// SIMATIC S7-200 project (STEP 7-Micro/WIN), CPU 224XP REL 02.01

ORGANIZATION_BLOCK 主程序:OB1
TITLE=程序注释
BEGIN
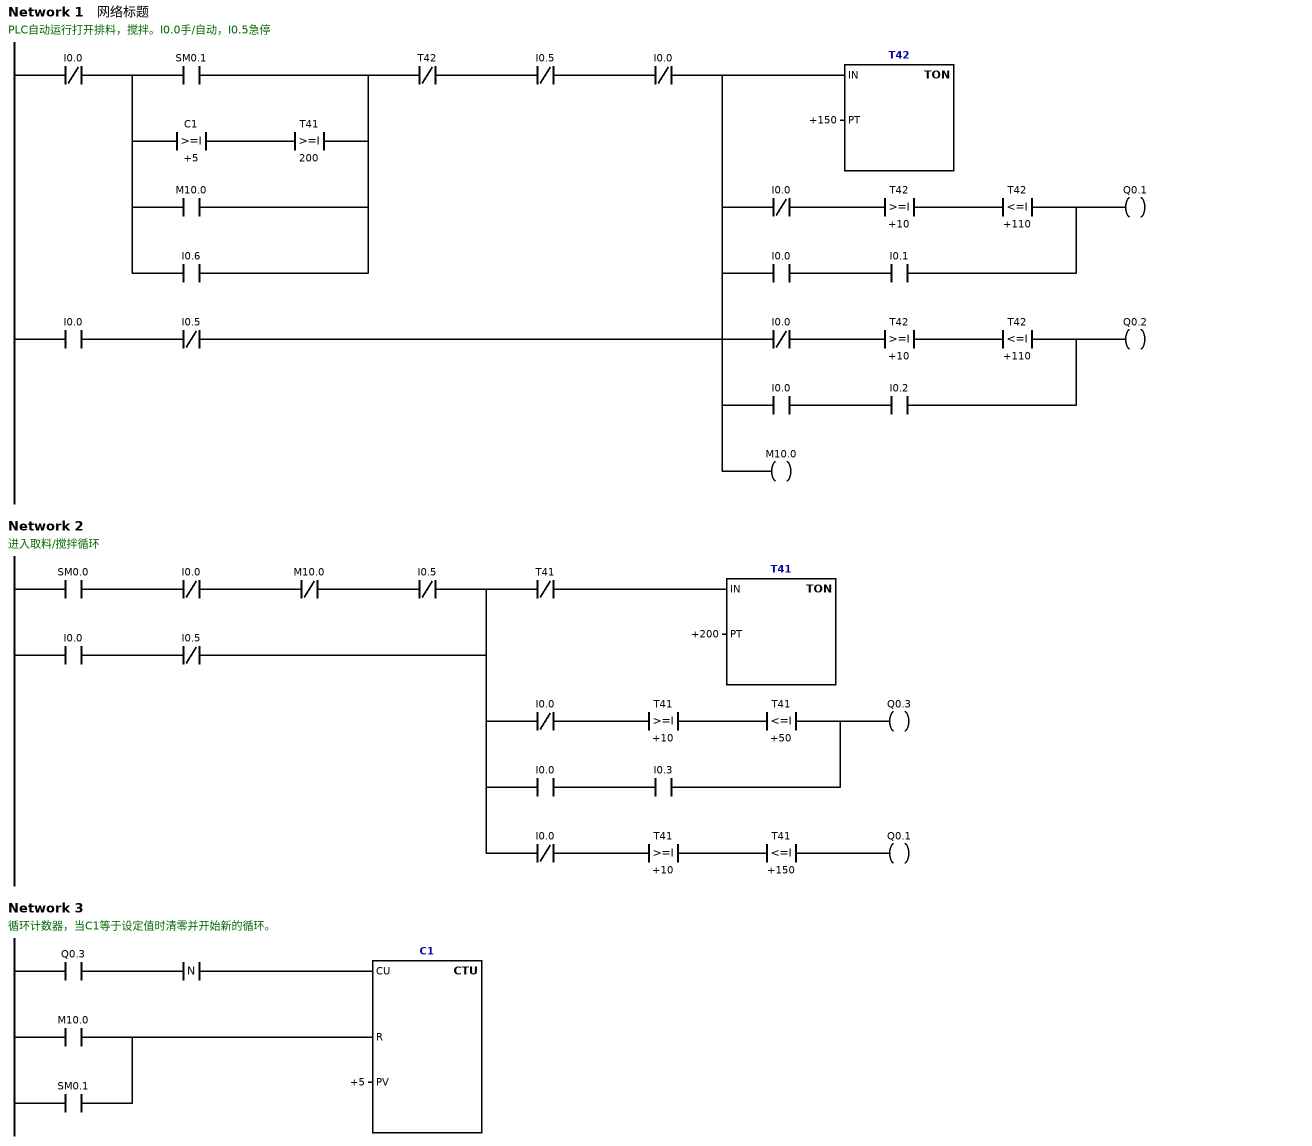
Network 1 //  网络标题
// PLC自动运行打开排料，搅拌。I0.0手/自动，I0.5急停
LDN    I0.0
LD     SM0.1
LDW>=  C1, +5
AW>=   T41, 200
OLD
O      M10.0
O      I0.6
ALD
AN     T42
AN     I0.5
AN     I0.0
LD     I0.0
AN     I0.5
OLD
LPS
TON    T42, +150
LDN    I0.0
AW>=   T42, +10
AW<=   T42, +110
LD     I0.0
A      I0.1
OLD
ALD
=      Q0.1
LRD
LDN    I0.0
AW>=   T42, +10
AW<=   T42, +110
LD     I0.0
A      I0.2
OLD
ALD
=      Q0.2
LPP
=      M10.0
Network 2
// 进入取料/搅拌循环
LD     SM0.0
AN     I0.0
AN     M10.0
AN     I0.5
LD     I0.0
AN     I0.5
OLD
LPS
AN     T41
TON    T41, +200
LRD
LDN    I0.0
AW>=   T41, +10
AW<=   T41, +50
LD     I0.0
A      I0.3
OLD
ALD
=      Q0.3
LPP
AN     I0.0
AW>=   T41, +10
AW<=   T41, +150
=      Q0.1
Network 3
// 循环计数器，当C1等于设定值时清零并开始新的循环。
LD     Q0.3
ED
LD     M10.0
O      SM0.1
CTU    C1, +5
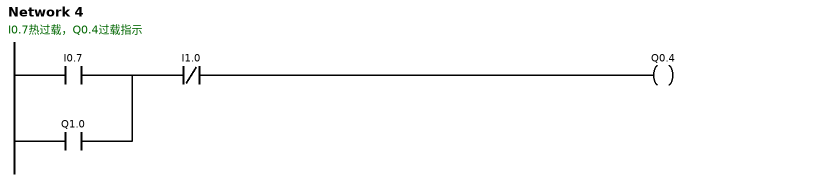
Network 4
// I0.7热过载，Q0.4过载指示
// (network saved uncompiled; LAD cells follow)
// row 0: c0 -| |- I0.7 v  c1 -|/|- I1.0  c2 --  c3 --  c4 --  c5 -( ) Q0.4
// row 1: c0 -| |- Q1.0 ^
END_ORGANIZATION_BLOCK
